// TIA Portal V16 export
// export: Created 2024-09-05T17:39:21.0739225Z, ExportSetting WithDefaults, DisplayName Totally Integrated Automation Portal, DisplayVersion V16 Update 6, DisplayName TIA Portal Version Control Interface, DisplayVersion V16 Update 2, DisplayName TIA Portal Openness, DisplayVersion V16 Update 6, DisplayName STEP 7 Professional, DisplayVersion V16 Update 6, DisplayName STEP 7 Safety, DisplayVersion V16, DisplayName WinCC Advanced, DisplayVersion V16 Update 6
FUNCTION_BLOCK "sq_jig"   // FB41, GRAPH
VERSION : 0.1
// stored: AcknowledgeErrorsRequired true, AutoNumber true, GraphVersion 6.0, InitialValuesAcquisition false, IsIECCheckEnabled false, LanguageInNetworks LAD, LockOperatingMode false, PermanentILProcessingInMANMode false, SetENOAutomatically false, SkipSteps false, UDAEnableTagReadback false, WithAlarmHandling true
   // inherited from GRAPH_BASE
   VAR
      OFF_SQ_BASE : Bool;
   END_VAR
   VAR_INPUT
      OFF_SQ { ExternalAccessible := 'False'; ExternalVisible := 'False'; ExternalWritable := 'False'} : Bool := false;   // Turn sequence off
      INIT_SQ { ExternalAccessible := 'False'; ExternalVisible := 'False'; ExternalWritable := 'False'} : Bool := false;   // Set sequence to initial state
      ACK_EF { ExternalAccessible := 'False'; ExternalVisible := 'False'; ExternalWritable := 'False'} : Bool := false;   // Acknowledge all errors and faults
      S_PREV { ExternalAccessible := 'False'; ExternalVisible := 'False'; ExternalWritable := 'False'} : Bool := false;   // Output previous step in parameter S_NO
      S_NEXT { ExternalAccessible := 'False'; ExternalVisible := 'False'; ExternalWritable := 'False'} : Bool := false;   // Indicate next step in parameter S_NO
      SW_AUTO { ExternalAccessible := 'False'; ExternalVisible := 'False'; ExternalWritable := 'False'} : Bool := false;   // Automatic mode
      SW_TAP { ExternalAccessible := 'False'; ExternalVisible := 'False'; ExternalWritable := 'False'} : Bool := false;   // Semiautomatic/switch with transition
      SW_TOP { ExternalAccessible := 'False'; ExternalVisible := 'False'; ExternalWritable := 'False'} : Bool := false;   // Semiautomatic/ignore transition
      SW_MAN { ExternalAccessible := 'False'; ExternalVisible := 'False'; ExternalWritable := 'False'} : Bool := false;   // Manual mode
      S_SEL { ExternalAccessible := 'False'; ExternalVisible := 'False'; ExternalWritable := 'False'} : Int := 0;   // Select step to be output to S_NO
      S_ON { ExternalAccessible := 'False'; ExternalVisible := 'False'; ExternalWritable := 'False'} : Bool := false;   // Activate step indicated in S_NO
      S_OFF { ExternalAccessible := 'False'; ExternalVisible := 'False'; ExternalWritable := 'False'} : Bool := false;   // Deactivate step indicated S_NO
      T_PUSH { ExternalAccessible := 'False'; ExternalVisible := 'False'; ExternalWritable := 'False'} : Bool := false;   // Enable transition to switch in semi automatic mode
   END_VAR
   VAR_OUTPUT
      S_NO { ExternalAccessible := 'False'; ExternalVisible := 'False'; ExternalWritable := 'False'} : Int := 0;   // Step number
      S_MORE { ExternalAccessible := 'False'; ExternalVisible := 'False'; ExternalWritable := 'False'} : Bool := false;   // More steps are available and can be shown in S_NO
      S_ACTIVE { ExternalAccessible := 'False'; ExternalVisible := 'False'; ExternalWritable := 'False'} : Bool := false;   // Step indicated in S_NO is active
      ERR_FLT { ExternalAccessible := 'False'; ExternalVisible := 'False'; ExternalWritable := 'False'} : Bool := false;   // Interlock or supervision group error
      AUTO_ON { ExternalAccessible := 'False'; ExternalVisible := 'False'; ExternalWritable := 'False'} : Bool := false;   // Automatic mode is active
      TAP_ON { ExternalAccessible := 'False'; ExternalVisible := 'False'; ExternalWritable := 'False'} : Bool := false;   // Semiautomatic mode/step with transition enabled
      TOP_ON { ExternalAccessible := 'False'; ExternalVisible := 'False'; ExternalWritable := 'False'} : Bool := false;   // Semiautomatic mode/ignore transition enabled
      MAN_ON { ExternalAccessible := 'False'; ExternalVisible := 'False'; ExternalWritable := 'False'} : Bool := false;   // Manual mode is active
   END_VAR
   VAR
      dummy : Bool;
      start : Bool;
      base : Bool;
   END_VAR
   VAR_TEMP   // added for the SCL form of the ladder/FBD networks
      _w1 : Bool;
   END_VAR
BEGIN
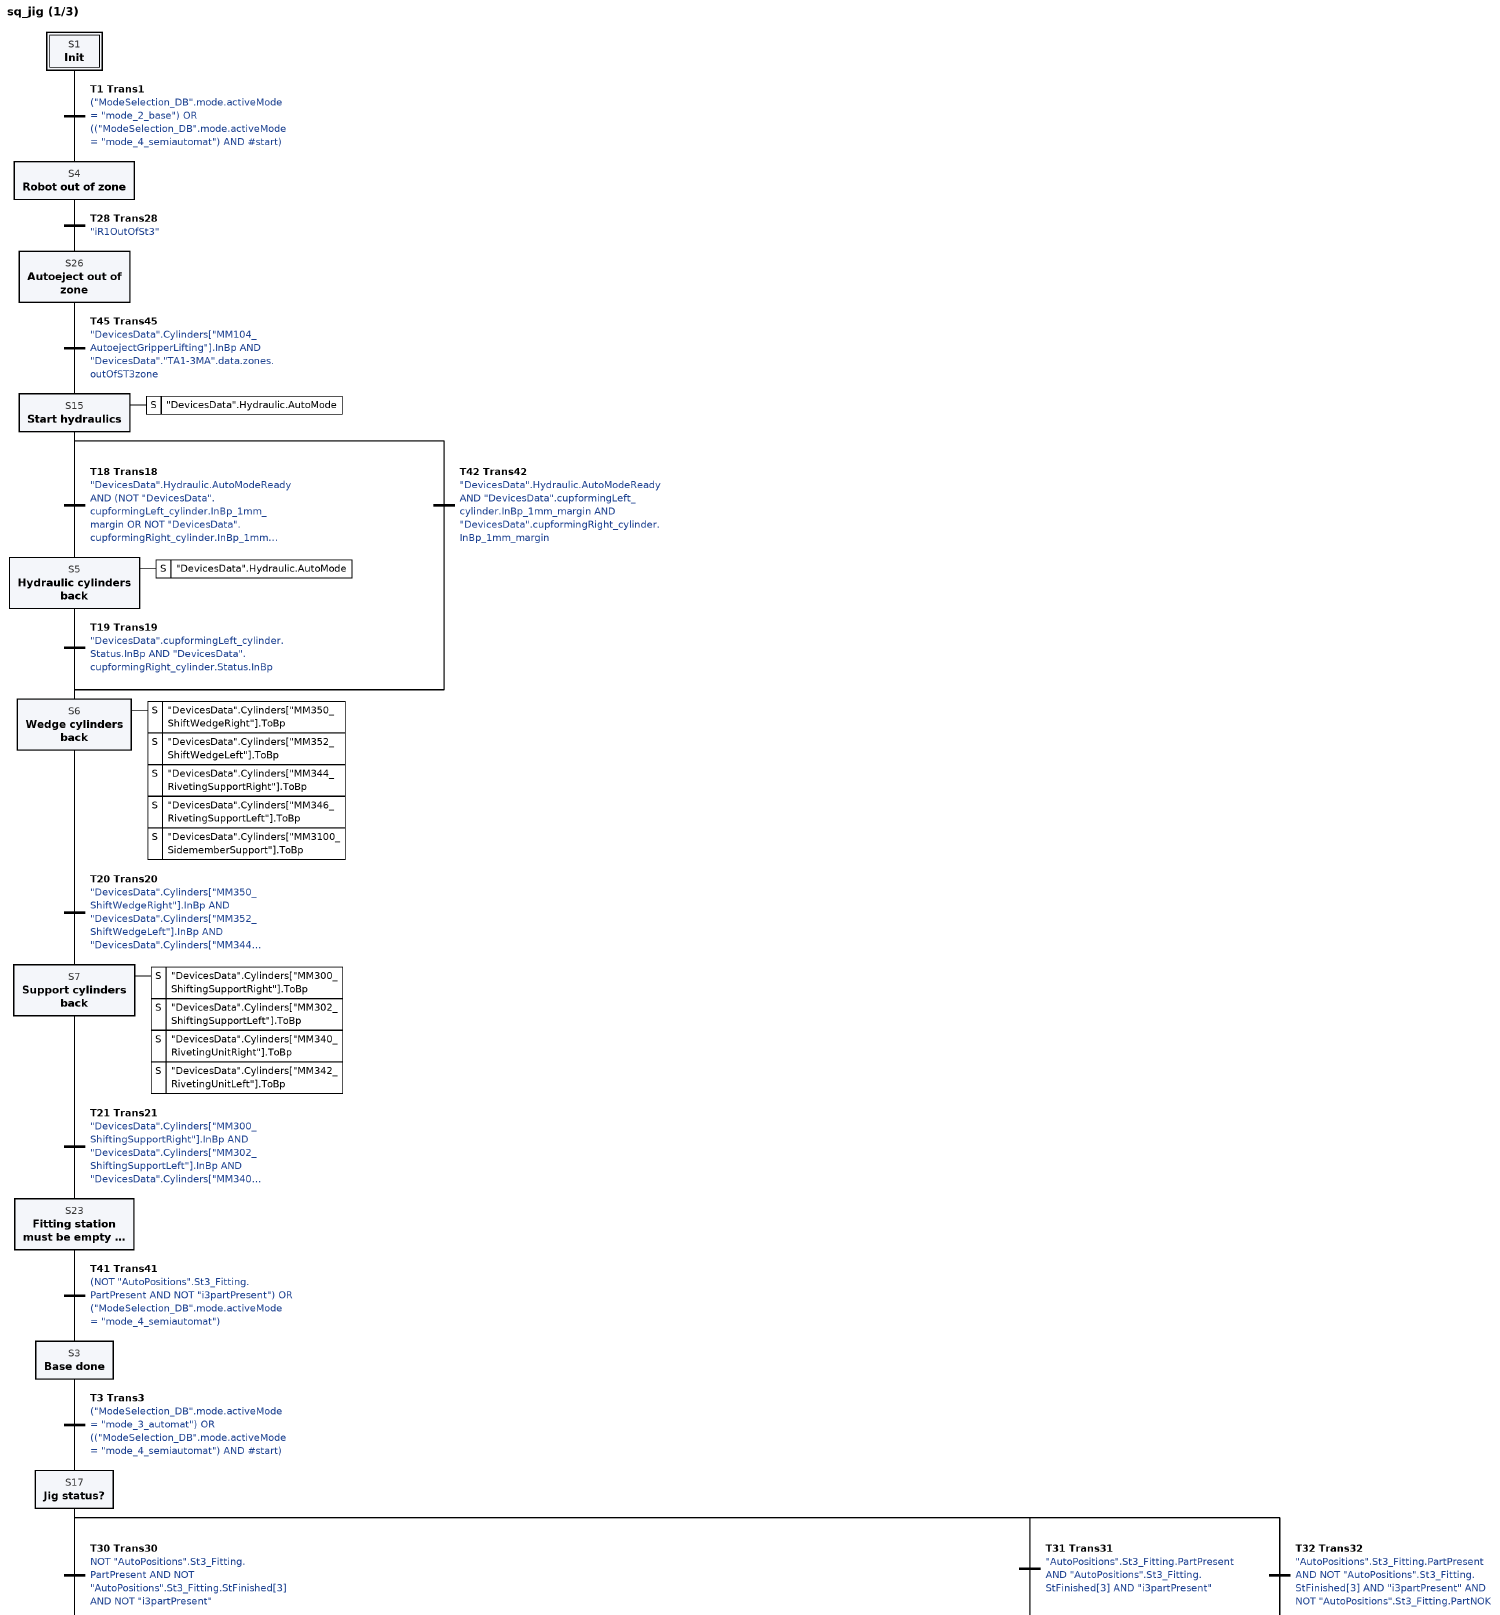
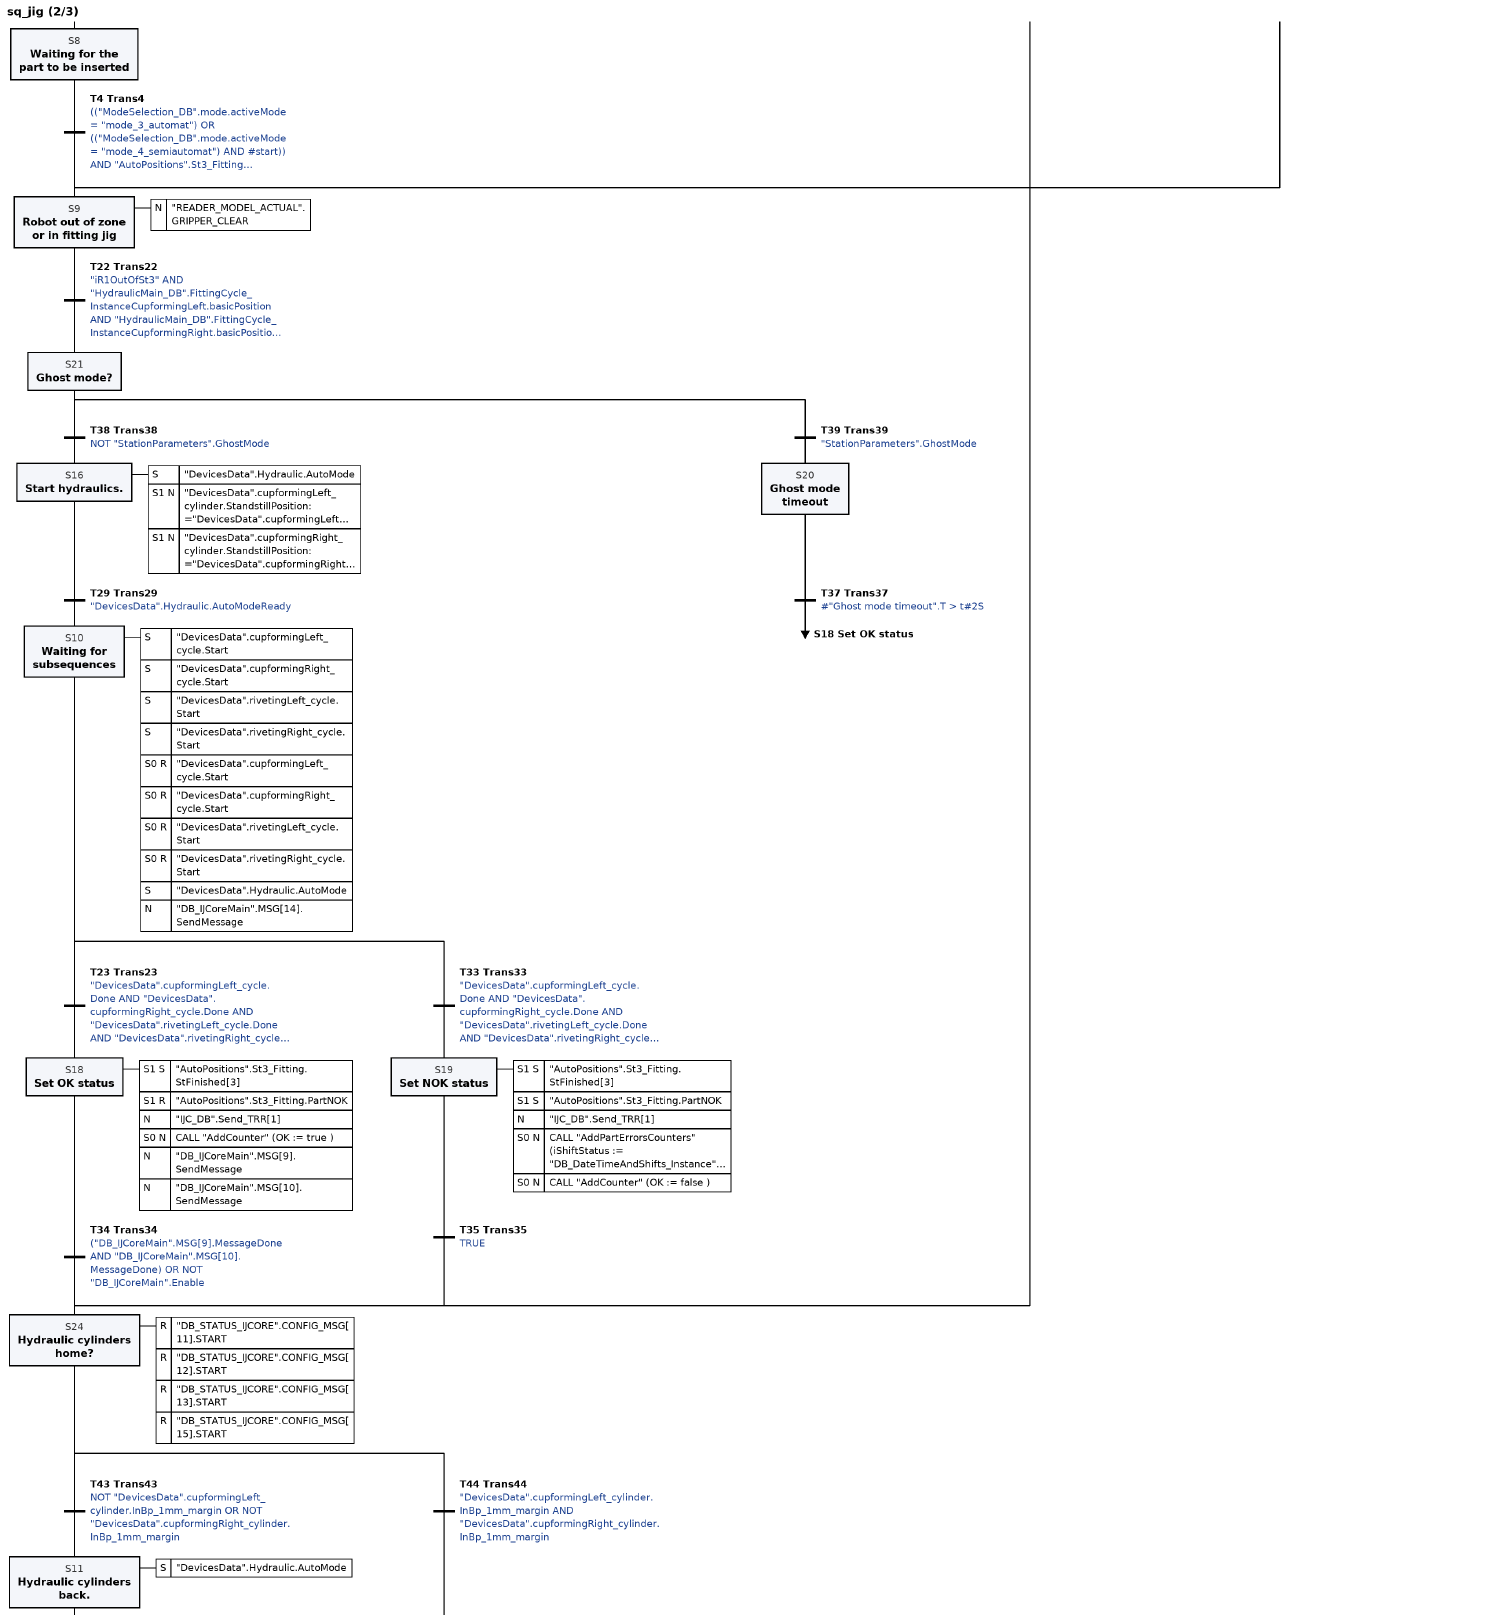
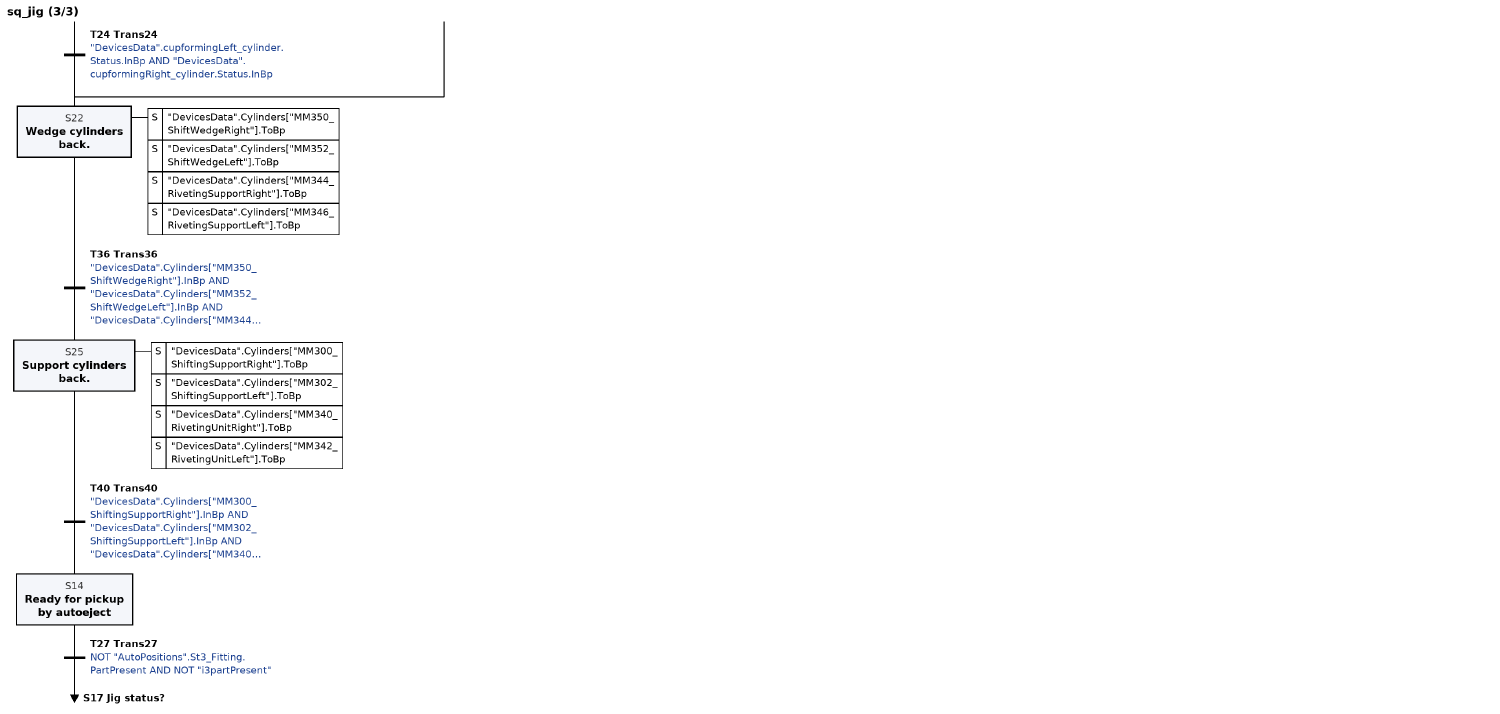
   // permanent pre-instructions
   NETWORK 1
   TITLE = base position
      #base := "HydraulicMain_DB".FittingCycle_InstanceCupformingLeft.basicPosition AND "HydraulicMain_DB".FittingCycle_InstanceCupformingRight.basicPosition AND "DB_Devices_Instance".RivetingCycleLeft_Instance.basicPosition AND "DB_Devices_Instance".RivetingCycleRight_Instance.basicPosition AND "DevicesData".Digiforce1.Ready AND "DevicesData".Digiforce1.programOK AND "DevicesData".Digiforce2.Ready AND "DevicesData".Digiforce2.programOK AND NOT "Devices_Diagnostic_DB".PNmissing;

   // sequencer 1
   INITIAL_STEP Init:   // S1, max time T#10S, warning time T#7S
   END_STEP
   TRANSITION Trans1 FROM Init TO "Robot out of zone"   // T1
      := ("ModeSelection_DB".mode.activeMode = "mode_2_base") OR (("ModeSelection_DB".mode.activeMode = "mode_4_semiautomat") AND #start);
   END_TRANSITION
   STEP "Start hydraulics":   // S15, max time T#10S, warning time T#7S
      supervision V := #"Start hydraulics".T > #"Start hydraulics".T_MAX;
              S    "DevicesData".Hydraulic.AutoMode
   END_STEP
   TRANSITION Trans18 FROM "Start hydraulics" TO "Hydraulic cylinders back"   // T18
      := "DevicesData".Hydraulic.AutoModeReady AND (NOT "DevicesData".cupformingLeft_cylinder.InBp_1mm_margin OR NOT "DevicesData".cupformingRight_cylinder.InBp_1mm_margin);
   END_TRANSITION
   TRANSITION Trans42 FROM "Start hydraulics" TO "Wedge cylinders back"   // T42
      := "DevicesData".Hydraulic.AutoModeReady AND "DevicesData".cupformingLeft_cylinder.InBp_1mm_margin AND "DevicesData".cupformingRight_cylinder.InBp_1mm_margin;
   END_TRANSITION
   STEP "Waiting for the part to be inserted":   // S8, max time T#10S, warning time T#7S
   END_STEP
   TRANSITION Trans4 FROM "Waiting for the part to be inserted" TO "Robot out of zone or in fitting jig"   // T4
      := (("ModeSelection_DB".mode.activeMode = "mode_3_automat") OR (("ModeSelection_DB".mode.activeMode = "mode_4_semiautomat") AND #start)) AND "AutoPositions".St3_Fitting.PartPresent AND NOT "AutoPositions".St3_Fitting.StFinished[3] AND ("i3partPresent" OR "StationParameters".GhostMode);
   END_TRANSITION
   STEP "Robot out of zone":   // S4, max time T#10S, warning time T#7S
      supervision V := #"Robot out of zone".T > #"Robot out of zone".T_MAX;
   END_STEP
   TRANSITION Trans28 FROM "Robot out of zone" TO "Autoeject out of zone"   // T28
      := "iR1OutOfSt3";
   END_TRANSITION
   STEP "Hydraulic cylinders back":   // S5, max time T#10S, warning time T#7S
      supervision V := #"Hydraulic cylinders back".T > #"Hydraulic cylinders back".T_MAX;
              S    "DevicesData".Hydraulic.AutoMode
   END_STEP
   TRANSITION Trans19 FROM "Hydraulic cylinders back" TO "Wedge cylinders back"   // T19
      := "DevicesData".cupformingLeft_cylinder.Status.InBp AND "DevicesData".cupformingRight_cylinder.Status.InBp;
   END_TRANSITION
   STEP "Wedge cylinders back":   // S6, max time T#10S, warning time T#7S
      supervision V := #"Wedge cylinders back".T > #"Wedge cylinders back".T_MAX;
              S    "DevicesData".Cylinders["MM350_ShiftWedgeRight"].ToBp
              S    "DevicesData".Cylinders["MM352_ShiftWedgeLeft"].ToBp
              S    "DevicesData".Cylinders["MM344_RivetingSupportRight"].ToBp
              S    "DevicesData".Cylinders["MM346_RivetingSupportLeft"].ToBp
              S    "DevicesData".Cylinders["MM3100_SidememberSupport"].ToBp
   END_STEP
   TRANSITION Trans20 FROM "Wedge cylinders back" TO "Support cylinders back"   // T20
      := "DevicesData".Cylinders["MM350_ShiftWedgeRight"].InBp AND "DevicesData".Cylinders["MM352_ShiftWedgeLeft"].InBp AND "DevicesData".Cylinders["MM344_RivetingSupportRight"].InBp AND "DevicesData".Cylinders["MM346_RivetingSupportLeft"].InBp AND "DevicesData".Cylinders["MM3100_SidememberSupport"].InBp;
   END_TRANSITION
   STEP "Support cylinders back":   // S7, max time T#10S, warning time T#7S
      supervision V := #"Support cylinders back".T > #"Support cylinders back".T_MAX;
              S    "DevicesData".Cylinders["MM300_ShiftingSupportRight"].ToBp
              S    "DevicesData".Cylinders["MM302_ShiftingSupportLeft"].ToBp
              S    "DevicesData".Cylinders["MM340_RivetingUnitRight"].ToBp
              S    "DevicesData".Cylinders["MM342_RivetingUnitLeft"].ToBp
   END_STEP
   TRANSITION Trans21 FROM "Support cylinders back" TO "Fitting station must be empty - remove part and delete status"   // T21
      := "DevicesData".Cylinders["MM300_ShiftingSupportRight"].InBp AND "DevicesData".Cylinders["MM302_ShiftingSupportLeft"].InBp AND "DevicesData".Cylinders["MM340_RivetingUnitRight"].InBp AND "DevicesData".Cylinders["MM342_RivetingUnitLeft"].InBp;
   END_TRANSITION
   STEP "Base done":   // S3, max time T#10S, warning time T#7S
   END_STEP
   TRANSITION Trans3 FROM "Base done" TO "Jig status?"   // T3
      := ("ModeSelection_DB".mode.activeMode = "mode_3_automat") OR (("ModeSelection_DB".mode.activeMode = "mode_4_semiautomat") AND #start);
   END_TRANSITION
   STEP "Robot out of zone or in fitting jig":   // S9, max time T#10S, warning time T#7S
      supervision V := #"Robot out of zone or in fitting jig".T > #"Robot out of zone or in fitting jig".T_MAX;
              N    "READER_MODEL_ACTUAL".GRIPPER_CLEAR
   END_STEP
   TRANSITION Trans22 FROM "Robot out of zone or in fitting jig" TO "Ghost mode?"   // T22
      := "iR1OutOfSt3" AND "HydraulicMain_DB".FittingCycle_InstanceCupformingLeft.basicPosition AND "HydraulicMain_DB".FittingCycle_InstanceCupformingRight.basicPosition AND "DB_Devices_Instance".RivetingCycleLeft_Instance.basicPosition AND "DB_Devices_Instance".RivetingCycleRight_Instance.basicPosition;
   END_TRANSITION
   STEP "Waiting for subsequences":   // S10, max time T#10S, warning time T#7S
              S    "DevicesData".cupformingLeft_cycle.Start
              S    "DevicesData".cupformingRight_cycle.Start
              S    "DevicesData".rivetingLeft_cycle.Start
              S    "DevicesData".rivetingRight_cycle.Start
          S0  R    "DevicesData".cupformingLeft_cycle.Start
          S0  R    "DevicesData".cupformingRight_cycle.Start
          S0  R    "DevicesData".rivetingLeft_cycle.Start
          S0  R    "DevicesData".rivetingRight_cycle.Start
              S    "DevicesData".Hydraulic.AutoMode
              N    "DB_IJCoreMain".MSG[14].SendMessage
   END_STEP
   TRANSITION Trans23 FROM "Waiting for subsequences" TO "Set OK status"   // T23
      := "DevicesData".cupformingLeft_cycle.Done AND "DevicesData".cupformingRight_cycle.Done AND "DevicesData".rivetingLeft_cycle.Done AND "DevicesData".rivetingRight_cycle.Done AND "DevicesData".cupformingLeft_cycle.OK AND "DevicesData".cupformingRight_cycle.OK AND "DevicesData".rivetingLeft_cycle.OK AND "DevicesData".rivetingRight_cycle.OK AND (("DB_IJCoreMain".MSG[14].MessageDone AND "DB_IJCoreMain".MSG[13].MessageDone AND ("DB_IJCoreMain".MSG[12].MessageDone OR "AlwaysTRUE")) OR NOT "DB_IJCoreMain".Enable) AND ("DB_IJCoreMain".MSG[15].MessageDone OR NOT "READER_MODEL_ACTUAL".PRODUCTO.NUM_TUBE);
   END_TRANSITION
   TRANSITION Trans33 FROM "Waiting for subsequences" TO "Set NOK status"   // T33
      := "DevicesData".cupformingLeft_cycle.Done AND "DevicesData".cupformingRight_cycle.Done AND "DevicesData".rivetingLeft_cycle.Done AND "DevicesData".rivetingRight_cycle.Done AND (("DB_IJCoreMain".MSG[14].MessageDone AND "DB_IJCoreMain".MSG[13].MessageDone AND ("DB_IJCoreMain".MSG[12].MessageDone OR "AlwaysTRUE")) OR NOT "DB_IJCoreMain".Enable) AND ("DB_IJCoreMain".MSG[15].MessageDone OR NOT "READER_MODEL_ACTUAL".PRODUCTO.NUM_TUBE);
   END_TRANSITION
   STEP "Hydraulic cylinders back.":   // S11, max time T#10S, warning time T#7S
      supervision V := #"Hydraulic cylinders back.".T > #"Hydraulic cylinders back.".T_MAX;
              S    "DevicesData".Hydraulic.AutoMode
   END_STEP
   TRANSITION Trans24 FROM "Hydraulic cylinders back." TO "Wedge cylinders back."   // T24
      := "DevicesData".cupformingLeft_cylinder.Status.InBp AND "DevicesData".cupformingRight_cylinder.Status.InBp;
   END_TRANSITION
   STEP "Autoeject out of zone":   // S26, max time T#10S, warning time T#7S
      supervision V := #"Autoeject out of zone".T > #"Autoeject out of zone".T_MAX;
   END_STEP
   TRANSITION Trans45 FROM "Autoeject out of zone" TO "Start hydraulics"   // T45
      := "DevicesData".Cylinders["MM104_AutoejectGripperLifting"].InBp AND "DevicesData"."TA1-3MA".data.zones.outOfST3zone;
   END_TRANSITION
   STEP "Ready for pickup by autoeject":   // S14, max time T#10S, warning time T#7S
   END_STEP
   TRANSITION Trans27 FROM "Ready for pickup by autoeject" TO "Jig status?"   // T27, jump
      := NOT "AutoPositions".St3_Fitting.PartPresent AND NOT "i3partPresent";
   END_TRANSITION
   STEP "Start hydraulics.":   // S16, max time T#10S, warning time T#7S
      supervision V := #"Start hydraulics.".T > #"Start hydraulics.".T_MAX;
              S    "DevicesData".Hydraulic.AutoMode
          S1  N    "DevicesData".cupformingLeft_cylinder.StandstillPosition:="DevicesData".cupformingLeft_cylinder.Position
          S1  N    "DevicesData".cupformingRight_cylinder.StandstillPosition:="DevicesData".cupformingRight_cylinder.Position
   END_STEP
   TRANSITION Trans29 FROM "Start hydraulics." TO "Waiting for subsequences"   // T29
      := "DevicesData".Hydraulic.AutoModeReady;
   END_TRANSITION
   STEP "Jig status?":   // S17, max time T#10S, warning time T#7S
   END_STEP
   TRANSITION Trans30 FROM "Jig status?" TO "Waiting for the part to be inserted"   // T30
      := NOT "AutoPositions".St3_Fitting.PartPresent AND NOT "AutoPositions".St3_Fitting.StFinished[3] AND NOT "i3partPresent";
   END_TRANSITION
   TRANSITION Trans31 FROM "Jig status?" TO "Hydraulic cylinders home?"   // T31
      := "AutoPositions".St3_Fitting.PartPresent AND "AutoPositions".St3_Fitting.StFinished[3] AND "i3partPresent";
   END_TRANSITION
   TRANSITION Trans32 FROM "Jig status?" TO "Robot out of zone or in fitting jig"   // T32
      := "AutoPositions".St3_Fitting.PartPresent AND NOT "AutoPositions".St3_Fitting.StFinished[3] AND "i3partPresent" AND NOT "AutoPositions".St3_Fitting.PartNOK;
   END_TRANSITION
   STEP "Set OK status":   // S18, max time T#10S, warning time T#7S
          S1  S    "AutoPositions".St3_Fitting.StFinished[3]
          S1  R    "AutoPositions".St3_Fitting.PartNOK
              N    "IJC_DB".Send_TRR[1]
          S0  N    CALL "AddCounter"
                   (OK := true
                   )
              N    "DB_IJCoreMain".MSG[9].SendMessage
              N    "DB_IJCoreMain".MSG[10].SendMessage
   END_STEP
   TRANSITION Trans34 FROM "Set OK status" TO "Hydraulic cylinders home?"   // T34
      := ("DB_IJCoreMain".MSG[9].MessageDone AND "DB_IJCoreMain".MSG[10].MessageDone) OR NOT "DB_IJCoreMain".Enable;
   END_TRANSITION
   STEP "Set NOK status":   // S19, max time T#10S, warning time T#7S
          S1  S    "AutoPositions".St3_Fitting.StFinished[3]
          S1  S    "AutoPositions".St3_Fitting.PartNOK
              N    "IJC_DB".Send_TRR[1]
          S0  N    CALL "AddPartErrorsCounters" (iShiftStatus := "DB_DateTimeAndShifts_Instance".ShiftStatus
                   )
          S0  N    CALL "AddCounter"
                   (OK := false
                   )
   END_STEP
   TRANSITION Trans35 FROM "Set NOK status" TO "Hydraulic cylinders home?"   // T35
      := TRUE;
   END_TRANSITION
   STEP "Ghost mode?":   // S21, max time T#10S, warning time T#7S
   END_STEP
   TRANSITION Trans38 FROM "Ghost mode?" TO "Start hydraulics."   // T38
      := NOT "StationParameters".GhostMode;
   END_TRANSITION
   TRANSITION Trans39 FROM "Ghost mode?" TO "Ghost mode timeout"   // T39
      := "StationParameters".GhostMode;
   END_TRANSITION
   STEP "Ghost mode timeout":   // S20, max time T#10S, warning time T#7S
   END_STEP
   TRANSITION Trans37 FROM "Ghost mode timeout" TO "Set OK status"   // T37, jump
      := #"Ghost mode timeout".T > t#2S;
   END_TRANSITION
   STEP "Fitting station must be empty - remove part and delete status":   // S23, max time T#2S, warning time T#7S
      supervision V := #"Fitting station must be empty - remove part and delete status".T > #"Fitting station must be empty - remove part and delete status".T_MAX;
   END_STEP
   TRANSITION Trans41 FROM "Fitting station must be empty - remove part and delete status" TO "Base done"   // T41
      := (NOT "AutoPositions".St3_Fitting.PartPresent AND NOT "i3partPresent") OR ("ModeSelection_DB".mode.activeMode = "mode_4_semiautomat");
   END_TRANSITION
   STEP "Hydraulic cylinders home?":   // S24, max time T#10S, warning time T#7S
              R    "DB_STATUS_IJCORE".CONFIG_MSG[11].START
              R    "DB_STATUS_IJCORE".CONFIG_MSG[12].START
              R    "DB_STATUS_IJCORE".CONFIG_MSG[13].START
              R    "DB_STATUS_IJCORE".CONFIG_MSG[15].START
   END_STEP
   TRANSITION Trans43 FROM "Hydraulic cylinders home?" TO "Hydraulic cylinders back."   // T43
      := NOT "DevicesData".cupformingLeft_cylinder.InBp_1mm_margin OR NOT "DevicesData".cupformingRight_cylinder.InBp_1mm_margin;
   END_TRANSITION
   TRANSITION Trans44 FROM "Hydraulic cylinders home?" TO "Wedge cylinders back."   // T44
      := "DevicesData".cupformingLeft_cylinder.InBp_1mm_margin AND "DevicesData".cupformingRight_cylinder.InBp_1mm_margin;
   END_TRANSITION
   STEP "Wedge cylinders back.":   // S22, max time T#10S, warning time T#7S
      supervision V := #"Wedge cylinders back.".T > #"Wedge cylinders back.".T_MAX;
              S    "DevicesData".Cylinders["MM350_ShiftWedgeRight"].ToBp
              S    "DevicesData".Cylinders["MM352_ShiftWedgeLeft"].ToBp
              S    "DevicesData".Cylinders["MM344_RivetingSupportRight"].ToBp
              S    "DevicesData".Cylinders["MM346_RivetingSupportLeft"].ToBp
   END_STEP
   TRANSITION Trans36 FROM "Wedge cylinders back." TO "Support cylinders back."   // T36
      := "DevicesData".Cylinders["MM350_ShiftWedgeRight"].InBp AND "DevicesData".Cylinders["MM352_ShiftWedgeLeft"].InBp AND "DevicesData".Cylinders["MM344_RivetingSupportRight"].InBp AND "DevicesData".Cylinders["MM346_RivetingSupportLeft"].InBp;
   END_TRANSITION
   STEP "Support cylinders back.":   // S25, max time T#10S, warning time T#7S
      supervision V := #"Support cylinders back.".T > #"Support cylinders back.".T_MAX;
              S    "DevicesData".Cylinders["MM300_ShiftingSupportRight"].ToBp
              S    "DevicesData".Cylinders["MM302_ShiftingSupportLeft"].ToBp
              S    "DevicesData".Cylinders["MM340_RivetingUnitRight"].ToBp
              S    "DevicesData".Cylinders["MM342_RivetingUnitLeft"].ToBp
   END_STEP
   TRANSITION Trans40 FROM "Support cylinders back." TO "Ready for pickup by autoeject"   // T40
      := "DevicesData".Cylinders["MM300_ShiftingSupportRight"].InBp AND "DevicesData".Cylinders["MM302_ShiftingSupportLeft"].InBp AND "DevicesData".Cylinders["MM340_RivetingUnitRight"].InBp AND "DevicesData".Cylinders["MM342_RivetingUnitLeft"].InBp;
   END_TRANSITION

   // permanent post-instructions
   NETWORK 1
   TITLE = Hydraulic cylinders back
      #_w1 := #"Hydraulic cylinders back".X OR #"Hydraulic cylinders back.".X;
      IF #_w1 AND NOT "DevicesData".cupformingLeft_cylinder.Status.InBp THEN
          "DevicesData".cupformingLeft_cylinder.Status.ToBp := TRUE;
      END_IF;
      IF #_w1 AND NOT "DevicesData".cupformingRight_cylinder.Status.InBp THEN
          "DevicesData".cupformingRight_cylinder.Status.ToBp := TRUE;
      END_IF;
      IF #_w1 AND "DevicesData".cupformingLeft_cylinder.Status.InBp THEN
          "DevicesData".cupformingLeft_cylinder.Status.ToBp := FALSE;
      END_IF;
      IF #_w1 AND "DevicesData".cupformingRight_cylinder.Status.InBp THEN
          "DevicesData".cupformingRight_cylinder.Status.ToBp := FALSE;
      END_IF;
END_FUNCTION_BLOCK
